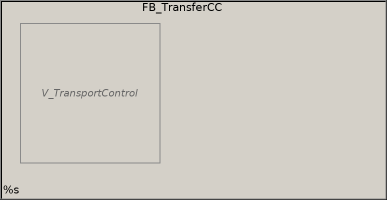
VISUALIZATION V_TransferCC  // 387x200
VAR_IN_OUT
	{attribute 'VAR_IN_OUT_AS_POINTER'}
	fbFunction		: FB_TransferCC;	
END_VAR
    Rectangle (0,0 387x200), colour toggle: fbFunction.BaseFunctionData.ZoneOrders[1].Drive_Run OR fbFunction.BaseFunctionData.ZoneOrders[1].Drive_RunRev
    Rectangle (0,180 200x20), "%s", text variable: fbFunction.ConfigFunction.FunctionName
    Label (139,0 107x15), "FB_TransferCC"
    Frame (20,23 140x140)
        shows V_TransportControl(TransportControl := fbFunction.fbTransportControl, ZoneData := fbFunction.ZoneData[1])
        p3560616238: SEL(fbFunction.HW_Inputs.Sensor_Pos_Left,SEL(fbFunction.HW_Inputs.Sensor_Pos_Right,100,0),200)
END_VISUALIZATION

(* stored: Version 1.1.0.1, ProductVersion 3.1.4024.9
   Visu V_TransferCC: Id {aa93d281-fc89-4afe-830c-d2ebddc63a18} *)
